{attribute 'qualified_only'}
VAR_GLOBAL INTERNAL
	debugMsg: ARRAY[1..Param.DEBUG_CAP] OF _DebugInfo;	
	nLastIdx: UDINT;
	
	nTotalNumber: UDINT;
	nNotifyNumber: UDINT;
	nPanicNumber: UDINT;
END_VAR

(* stored: Version 1.1.0.1
   GVL _Debug: Id {c602205e-748f-438e-a90c-f30a653e50a0} *)
